{attribute 'qualified_only'}
VAR_GLOBAL
	 stTimer2 : ST_timer := (tTimer := T#5S); 
END_VAR

(* stored: Version 1.1.0.1, ProductVersion 3.1.4024.12
   GVL G_task2: Id {23487ebd-7a32-4586-9594-69091bf7ec75} *)
